PROGRAM P_StationUnloadFrock_L
VAR
	_station:					REFERENCE TO ST_SystemStation;
	_bEnable: 					BOOL;
	
	_bManual:                   BOOL;//  手动下料
END_VAR

_station REF= G_arrStation[E_Station.UnloadFrock_L];
_station.arrName[E_Language.Chinese]:="下工装线体";
_station.arrName[E_Language.Vietnamese]:="Thiết bị dây";
_bEnable:=NOT GVL.stSetting.arrStationShield[E_Station.UnloadFrock_L];

_bManual:=GVL.stSetting.bManualUnloadFrock;

A_Auto();
A_Home();

ACTION A_Auto:
CASE _station.iStepNow OF
	1000:
		_station.arrInfo[E_Language.Chinese]:="初始化完成等待启动";
		IF _bEnable THEN
			_station.iStepNext:=1101;
		END_IF
	1101:
		_station.arrInfo[E_Language.Chinese]:="判断是否有料";
		IF NOT GVL.I.bUnloadFrockConveyorCheck2 THEN
			_station.iStepNext:=1201;
		END_IF
	1201:
		_station.arrInfo[E_Language.Chinese]:="等待请求上料";
		IF GVL.stHandshake.bUnloadFrockToUnloadFrock_L THEN
			GVL.stHandshake.bUnloadFrock_LToUnloadFrock:=TRUE;
			_station.iStepNext:=1301;
		END_IF
	1301:
		_station.arrInfo[E_Language.Chinese]:="等待复位请求信号";
		IF NOT GVL.stHandshake.bUnloadFrockToUnloadFrock_L THEN
			GVL.stHandshake.bUnloadFrock_LToUnloadFrock:=FALSE;
			_station.iStepNext:=1401;
		END_IF
	1401:
		_station.arrInfo[E_Language.Chinese]:="等待产品到位";
		GVL.stOverTime.bUnloadFrockConveyorCheck2:=TRUE;
		IF GVL.I.bUnloadFrockConveyorCheck2 THEN
			GVL.stOverTime.bUnloadFrockConveyorCheck2:=FALSE;
			_station.iStepNext:=1451;
		END_IF
	1451:
		IF NOT _bManual  THEN
			_station.iStepNext:=1501;
			ELSE
			_station.iStepNext:=1101;
		END_IF
	1501:
		_station.arrInfo[E_Language.Chinese]:="升降气缸伸出";
		IF G_arrFbCylinder[E_Cylinder.UnloadFrockConveyorPrevent].M_WorkRequest() THEN
			_station.iStepNext:=1601;
		END_IF
	1601:
		_station.arrInfo[E_Language.Chinese]:="拨料气缸拨料";
		IF G_arrFbCylinder[E_Cylinder.UnloadFrockConveyorPush].M_WorkRequest() THEN
			_station.iStepNext:=1701;
		END_IF
	1701:
		_station.arrInfo[E_Language.Chinese]:="升降气缸缩回 拨料气缸缩回";
		IF  G_arrFbCylinder[E_Cylinder.UnloadFrockConveyorPush].M_HomeRequest() AND G_arrFbCylinder[E_Cylinder.UnloadFrockConveyorPrevent].M_HomeRequest() THEN
			_station.iStepNext:=1101;
		END_IF
END_CASE
END_ACTION

ACTION A_Home:
CASE _station.iStepNow OF
	0:
		_station.arrInfo[E_Language.Chinese]:="等待初始化";
		_station.iStepNext:=SEL(_bEnable,1000,100);
	100:
	    IF NOT _bManual  THEN
			_station.iStepNext:=200;
			ELSE
			_station.iStepNext:=1000;
		END_IF
	200:
		_station.arrInfo[E_Language.Chinese]:="升降气缸缩回";
		IF G_arrFbCylinder[E_Cylinder.UnloadFrockConveyorPrevent].M_HomeRequest() THEN
			_station.iStepNext:=300;
		END_IF
	300:
		_station.arrInfo[E_Language.Chinese]:="拨料气缸缩回";
		IF G_arrFbCylinder[E_Cylinder.UnloadFrockConveyorPush].M_HomeRequest() THEN
			_station.iStepNext:=1000;
		END_IF
END_CASE
END_ACTION

END_PROGRAM

(* stored: Version 1.1.0.1, ProductVersion 3.1.4024.3
   POU P_StationUnloadFrock_L: Id {b55114a8-92ae-4be8-986e-0682fb29b6b7}, SpecialFunc None
   Action A_Auto: Id {4934aa77-4ad8-4294-a961-fcf20b3634a4}
   Action A_Home: Id {67ad5919-61ea-4c19-8fd4-58ae50a211b2} *)
